FUNCTION_BLOCK FB_LTU_Cylinder
VAR
		bLightBarrier	AT %I*			: BOOL;				// LTU light sensor 
		bToBottom		AT %Q* 			: BOOL; 			// Output TO Bottom	
		bToTop			AT %Q* 			: BOOL; 			// Output To Top
		bAtBottom		AT %I*			: BOOL; 			//Input At Bottom 
		bAtMiddle 		AT %I* 			: BOOL; 			//Input At Middle	 
		bAtTop			AT %I* 			: BOOL; 			//Input At Top 
		LTU_Motor						: FB_ConveyorMotor;	//LTU Motor
END_VAR

PROPERTY AtBottom : BOOL
GET
AtBottom:= bAtBottom;
END_GET
END_PROPERTY

PROPERTY AtMiddle : BOOL
GET
AtMiddle:= bAtMiddle;
END_GET
END_PROPERTY

PROPERTY AtTop : BOOL
GET
AtTop:= bAtTop;
END_GET
END_PROPERTY

METHOD MoveBottom : BOOL
VAR
	Cylinder	:FB_LTU_Cylinder;
END_VAR
IF NOT Cylinder.Occupied THEN
Cylinder.ToBottom	:=TRUE; 	// Set Output To bottom to True 
Cylinder.ToTop	:=FALSE;		// Set Output To Top to FALSE
END_IF
IF NOT Cylinder.AtTop AND Cylinder.AtBottom AND NOT Cylinder.AtMiddle THEN //Check the feedback inputs
	MoveBottom:=TRUE;			//return true
	ELSE
		MoveBottom:=FALSE;		//return false
END_IF
END_METHOD

METHOD MoveMiddle : BOOL
VAR
	Cylinder	:FB_LTU_Cylinder;
END_VAR
IF NOT Cylinder.Occupied THEN
Cylinder.ToBottom	:=FALSE; 	// Set Output To bottom to false 
Cylinder.ToTop	:=FALSE;		// Set Output To Top to false
END_IF
IF NOT Cylinder.AtTop AND NOT Cylinder.AtBottom AND Cylinder.AtMiddle THEN //Check the feedback inputs
	MoveMiddle:=TRUE;			//return true
	ELSE
		MoveMiddle:=FALSE;		//return false
END_IF
END_METHOD

METHOD MoveTop : BOOL
VAR
	Cylinder	:FB_LTU_Cylinder;
END_VAR
IF NOT Cylinder.Occupied THEN
Cylinder.ToBottom	:=FALSE; 	// Set Output To bottom to false 
Cylinder.ToTop	:=TRUE;		// Set Output To Top to True
END_IF
IF Cylinder.AtTop AND NOT Cylinder.AtBottom AND NOT Cylinder.AtMiddle THEN
	MoveTop:=TRUE;
	ELSE
		MoveTop:=FALSE;
END_IF
END_METHOD

PROPERTY Occupied : BOOL
GET
Occupied:= bLightBarrier;
END_GET
END_PROPERTY

PROPERTY ToBottom : BOOL
SET
bToBottom:=ToBottom ;
END_SET
END_PROPERTY

PROPERTY ToTop : BOOL
SET
bToTop:=ToTop;
END_SET
END_PROPERTY

END_FUNCTION_BLOCK

(* stored: Version 1.1.0.1, ProductVersion 3.1.4024.12
   POU FB_LTU_Cylinder: Id {cc59b657-e855-4776-960f-eb7ca159d0ee}, SpecialFunc None
   Property AtBottom: Id {3bb3c766-0639-44a8-a2ae-822de9cac397}
   Get Get: Id {663dfa3f-b281-48c7-a740-923df32175a5}
   Property AtMiddle: Id {faf13aff-938b-4b0a-86be-4224b05306a6}
   Get Get: Id {04704a0b-7bd6-4d5f-b320-427439c8cd11}
   Property AtTop: Id {db968124-0667-4b0a-8874-81fed56a7cb8}
   Get Get: Id {44b3b79d-f45c-419a-a130-11ed20a1aee3}
   Method MoveBottom: Id {ec4556e9-625d-498a-9655-1896ff9c38f4}
   Method MoveMiddle: Id {ea84f625-db3b-4e66-8901-0e15008833f1}
   Method MoveTop: Id {0c213e24-7355-4c4b-b171-57858d42070d}
   Property Occupied: Id {9c4762a7-1f18-4268-aa4a-db629d522d37}
   Get Get: Id {4a1209fb-7c1a-43b2-aea6-88d80c1722e0}
   Property ToBottom: Id {76cfa9ed-fb63-4444-a972-559fc40806bc}
   Set Set: Id {045070d4-24c3-4e82-9e2a-e28760a5485d}
   Property ToTop: Id {0c97d193-059a-4ea1-a595-050f99df4e9a}
   Set Set: Id {cdd7e902-c458-42be-94a1-623620cc0ade} *)
